{attribute 'qualified_only'}
VAR_GLOBAL
	//Endstop
	bEndStopUpActive 				: BOOL;
	bEndStopDownActive 				: BOOL;
	bEndStopOverride 				: BOOL; 
	
	//Displacementcontrol
	bDisplacement_target_active		:BOOL;
	fProportionalgain				:LREAL := 1.0;
	fDisplacement_target			:LREAL;
END_VAR

(* stored: Version 1.1.0.1
   GVL HMI: Id {26f8b220-c366-427c-968e-e98e5cf6b52c} *)
